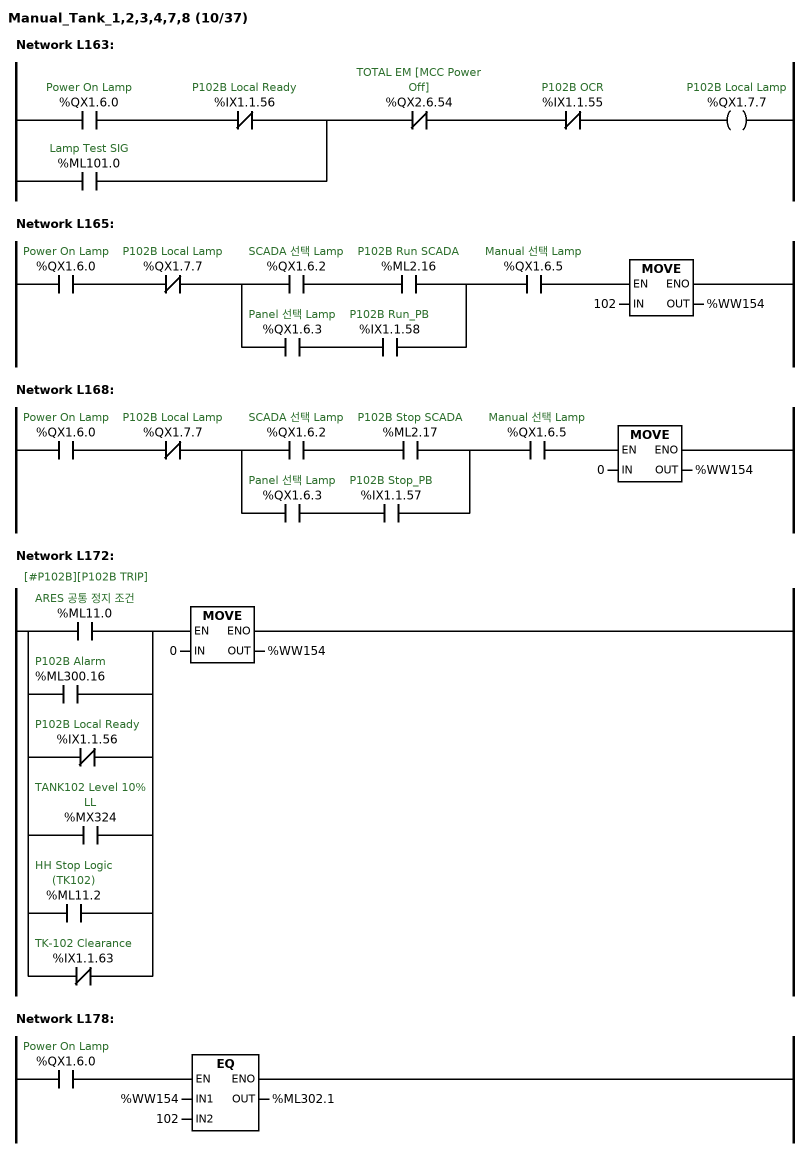
(* [picture p24: Manual_Tank_1,2,3,4,7,8 rungs L163-L178] *)
(* Rung L163 *)
%QX1.7.7 := ((%QX1.6.0 AND NOT %IX1.1.56) OR %ML101.0) AND NOT %QX2.6.54 AND NOT %IX1.1.55;
(* Rung L165 *)
IF %QX1.6.0 AND NOT %QX1.7.7 AND ((%QX1.6.2 AND %ML2.16) OR (%QX1.6.3 AND %IX1.1.58)) AND %QX1.6.5 THEN
    %WW154 := 102;
END_IF;
(* Rung L168 *)
IF %QX1.6.0 AND NOT %QX1.7.7 AND ((%QX1.6.2 AND %ML2.17) OR (%QX1.6.3 AND %IX1.1.57)) AND %QX1.6.5 THEN
    %WW154 := 0;
END_IF;
(* [#P102B][P102B TRIP] *)
(* Rung L172 *)
IF %ML11.0 OR %ML300.16 OR NOT %IX1.1.56 OR %MX324 OR %ML11.2 OR NOT %IX1.1.63 THEN %WW154 := 0; END_IF;
(* Rung L178 *)
IF %QX1.6.0 THEN %ML302.1 := %WW154 = 102; END_IF;

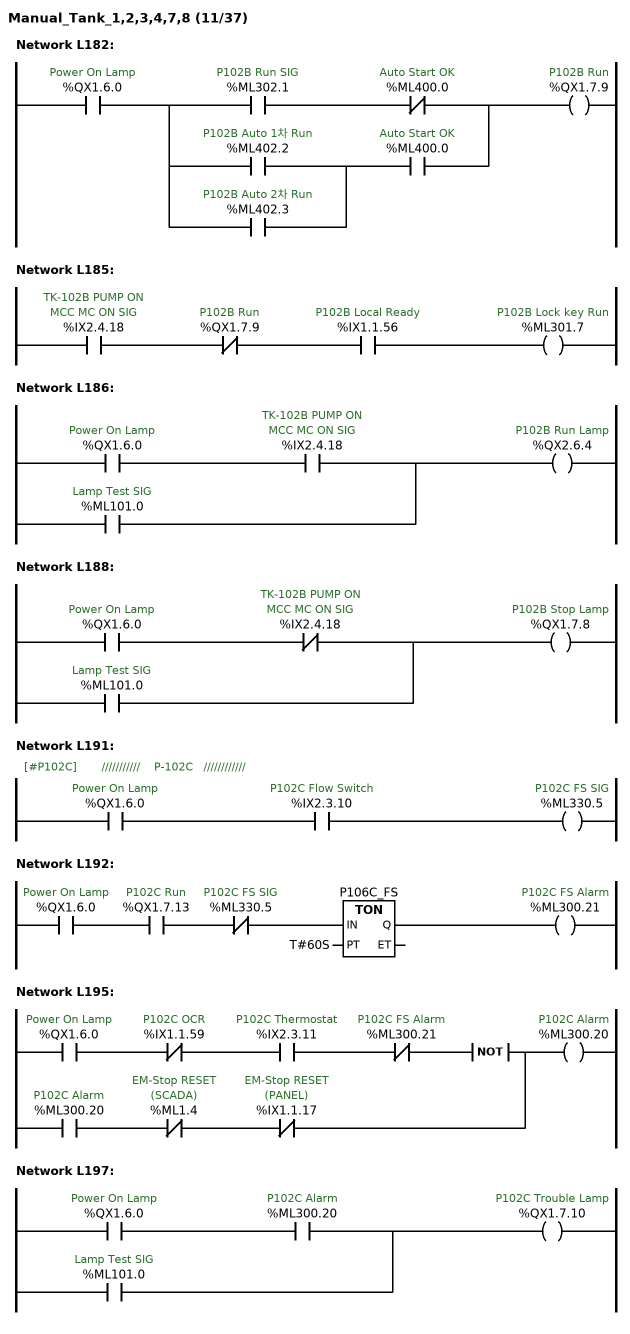
(* Rung L182 *)
%QX1.7.9 := %QX1.6.0 AND ((%ML302.1 AND NOT %ML400.0) OR ((%ML402.2 OR %ML402.3) AND %ML400.0));
(* Rung L185 *)
%ML301.7 := %IX2.4.18 AND NOT %QX1.7.9 AND %IX1.1.56;
(* Rung L186 *)
%QX2.6.4 := (%QX1.6.0 AND %IX2.4.18) OR %ML101.0;
(* Rung L188 *)
%QX1.7.8 := (%QX1.6.0 AND NOT %IX2.4.18) OR %ML101.0;
(* [#P102C]       ///////////    P-102C   //////////// *)
(* Rung L191 *)
%ML330.5 := %QX1.6.0 AND %IX2.3.10;
(* Rung L192 *)
P106C_FS(IN := %QX1.6.0 AND %QX1.7.13 AND NOT %ML330.5, PT := T#60S);
%ML300.21 := P106C_FS.Q;
(* Rung L195 *)
%ML300.20 := NOT (%QX1.6.0 AND NOT %IX1.1.59 AND %IX2.3.11 AND NOT %ML300.21) OR (%ML300.20 AND NOT %ML1.4 AND NOT %IX1.1.17);
(* Rung L197 *)
%QX1.7.10 := (%QX1.6.0 AND %ML300.20) OR %ML101.0;

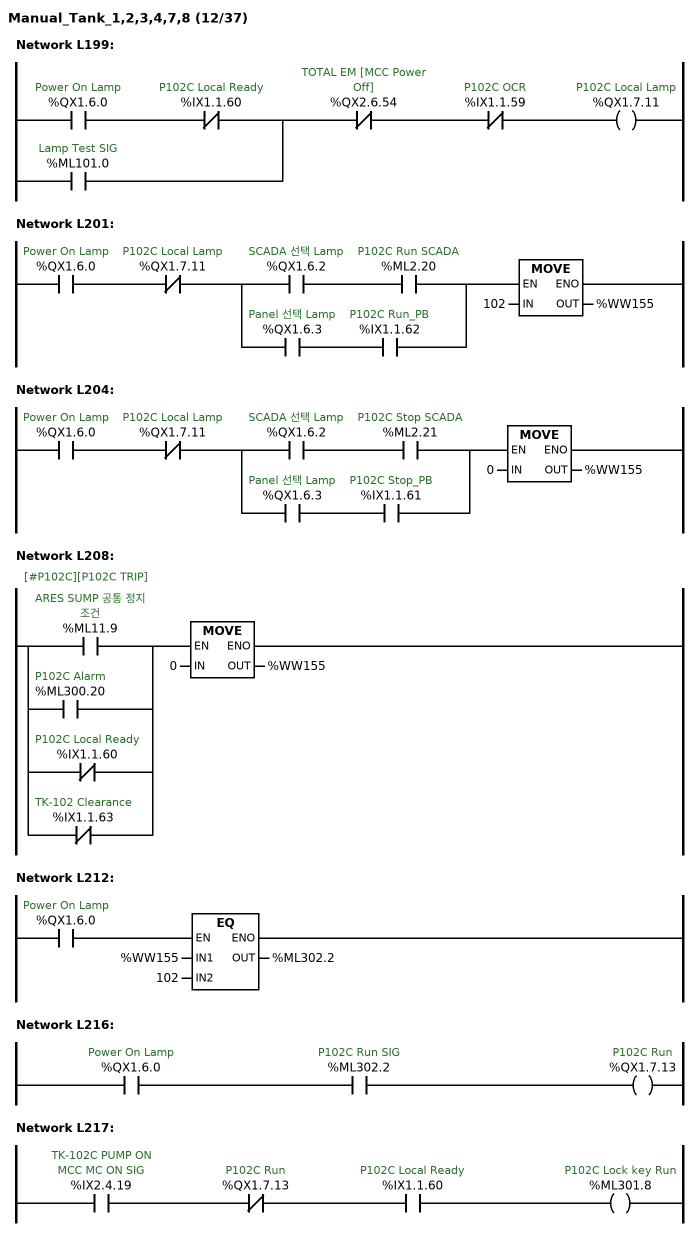
(* Rung L199 *)
%QX1.7.11 := ((%QX1.6.0 AND NOT %IX1.1.60) OR %ML101.0) AND NOT %QX2.6.54 AND NOT %IX1.1.59;
(* Rung L201 *)
IF %QX1.6.0 AND NOT %QX1.7.11 AND ((%QX1.6.2 AND %ML2.20) OR (%QX1.6.3 AND %IX1.1.62)) THEN
    %WW155 := 102;
END_IF;
(* Rung L204 *)
IF %QX1.6.0 AND NOT %QX1.7.11 AND ((%QX1.6.2 AND %ML2.21) OR (%QX1.6.3 AND %IX1.1.61)) THEN
    %WW155 := 0;
END_IF;
(* [#P102C][P102C TRIP] *)
(* Rung L208 *)
IF %ML11.9 OR %ML300.20 OR NOT %IX1.1.60 OR NOT %IX1.1.63 THEN %WW155 := 0; END_IF;
(* Rung L212 *)
IF %QX1.6.0 THEN %ML302.2 := %WW155 = 102; END_IF;
(* Rung L216 *)
%QX1.7.13 := %QX1.6.0 AND %ML302.2;
(* Rung L217 *)
%ML301.8 := %IX2.4.19 AND NOT %QX1.7.13 AND %IX1.1.60;

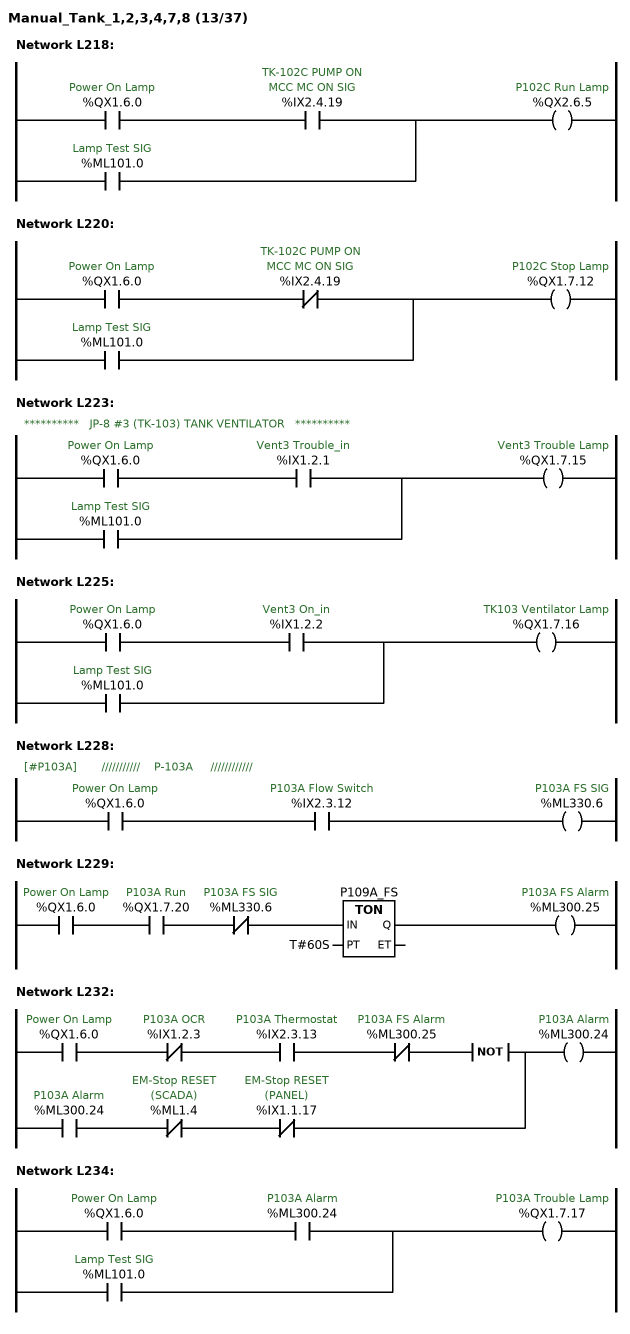
(* Rung L218 *)
%QX2.6.5 := (%QX1.6.0 AND %IX2.4.19) OR %ML101.0;
(* Rung L220 *)
%QX1.7.12 := (%QX1.6.0 AND NOT %IX2.4.19) OR %ML101.0;
(* **********   JP-8 #3 (TK-103) TANK VENTILATOR   ********** *)
(* Rung L223 *)
%QX1.7.15 := (%QX1.6.0 AND %IX1.2.1) OR %ML101.0;
(* Rung L225 *)
%QX1.7.16 := (%QX1.6.0 AND %IX1.2.2) OR %ML101.0;
(* [#P103A]       ///////////    P-103A     //////////// *)
(* Rung L228 *)
%ML330.6 := %QX1.6.0 AND %IX2.3.12;
(* Rung L229 *)
P109A_FS(IN := %QX1.6.0 AND %QX1.7.20 AND NOT %ML330.6, PT := T#60S);
%ML300.25 := P109A_FS.Q;
(* Rung L232 *)
%ML300.24 := NOT (%QX1.6.0 AND NOT %IX1.2.3 AND %IX2.3.13 AND NOT %ML300.25) OR (%ML300.24 AND NOT %ML1.4 AND NOT %IX1.1.17);
(* Rung L234 *)
%QX1.7.17 := (%QX1.6.0 AND %ML300.24) OR %ML101.0;

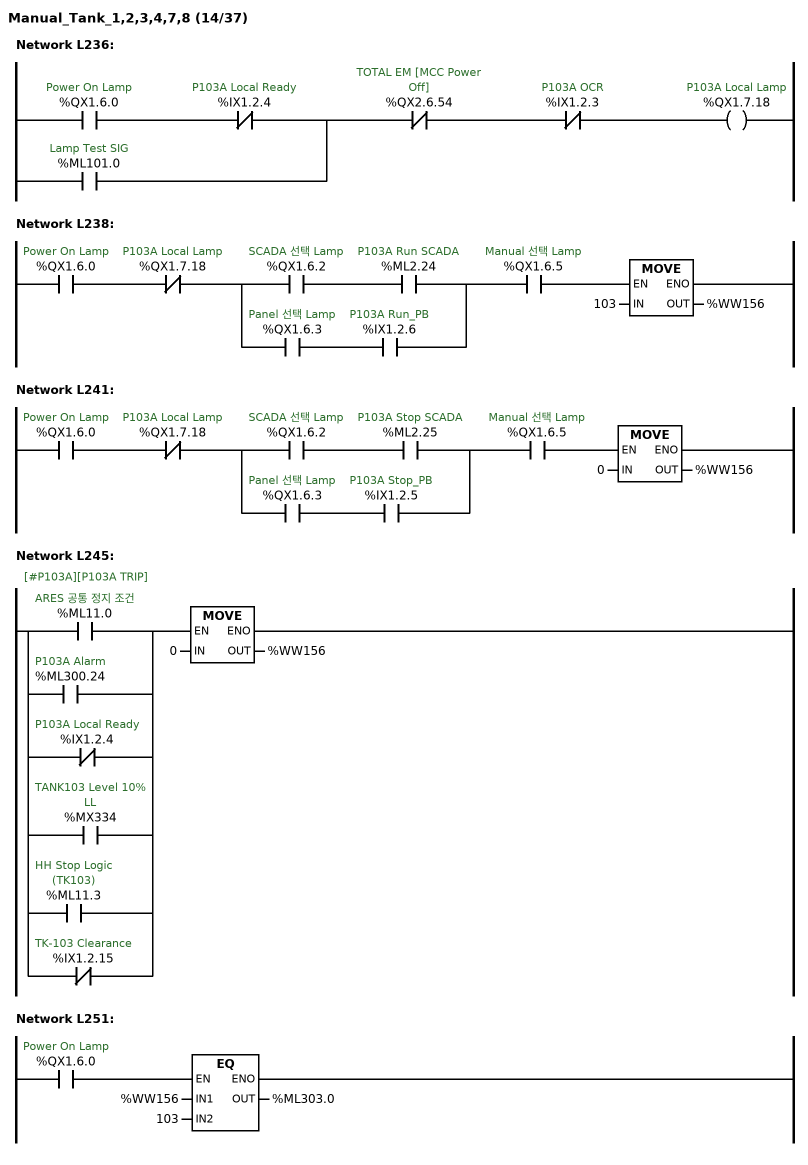
(* Rung L236 *)
%QX1.7.18 := ((%QX1.6.0 AND NOT %IX1.2.4) OR %ML101.0) AND NOT %QX2.6.54 AND NOT %IX1.2.3;
(* Rung L238 *)
IF %QX1.6.0 AND NOT %QX1.7.18 AND ((%QX1.6.2 AND %ML2.24) OR (%QX1.6.3 AND %IX1.2.6)) AND %QX1.6.5 THEN
    %WW156 := 103;
END_IF;
(* Rung L241 *)
IF %QX1.6.0 AND NOT %QX1.7.18 AND ((%QX1.6.2 AND %ML2.25) OR (%QX1.6.3 AND %IX1.2.5)) AND %QX1.6.5 THEN
    %WW156 := 0;
END_IF;
(* [#P103A][P103A TRIP] *)
(* Rung L245 *)
IF %ML11.0 OR %ML300.24 OR NOT %IX1.2.4 OR %MX334 OR %ML11.3 OR NOT %IX1.2.15 THEN %WW156 := 0; END_IF;
(* Rung L251 *)
IF %QX1.6.0 THEN %ML303.0 := %WW156 = 103; END_IF;

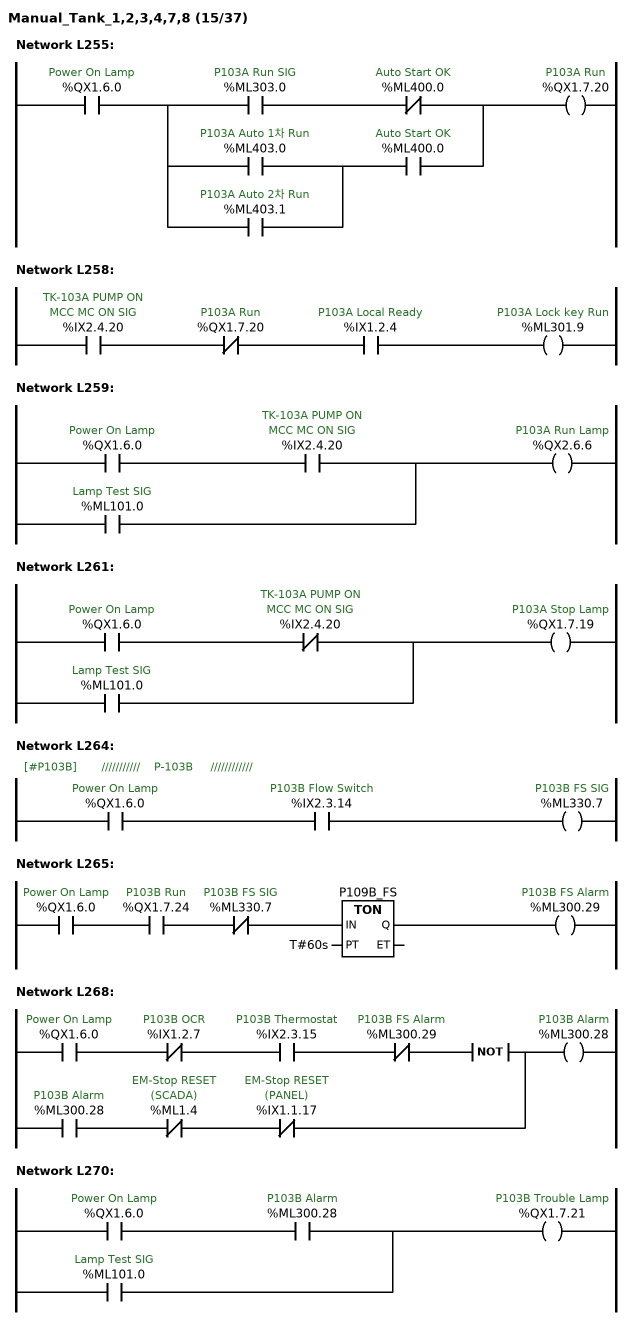
(* Rung L255 *)
%QX1.7.20 := %QX1.6.0 AND ((%ML303.0 AND NOT %ML400.0) OR ((%ML403.0 OR %ML403.1) AND %ML400.0));
(* Rung L258 *)
%ML301.9 := %IX2.4.20 AND NOT %QX1.7.20 AND %IX1.2.4;
(* Rung L259 *)
%QX2.6.6 := (%QX1.6.0 AND %IX2.4.20) OR %ML101.0;
(* Rung L261 *)
%QX1.7.19 := (%QX1.6.0 AND NOT %IX2.4.20) OR %ML101.0;
(* [#P103B]       ///////////    P-103B     //////////// *)
(* Rung L264 *)
%ML330.7 := %QX1.6.0 AND %IX2.3.14;
(* Rung L265 *)
P109B_FS(IN := %QX1.6.0 AND %QX1.7.24 AND NOT %ML330.7, PT := T#60s);
%ML300.29 := P109B_FS.Q;
(* Rung L268 *)
%ML300.28 := NOT (%QX1.6.0 AND NOT %IX1.2.7 AND %IX2.3.15 AND NOT %ML300.29) OR (%ML300.28 AND NOT %ML1.4 AND NOT %IX1.1.17);
(* Rung L270 *)
%QX1.7.21 := (%QX1.6.0 AND %ML300.28) OR %ML101.0;

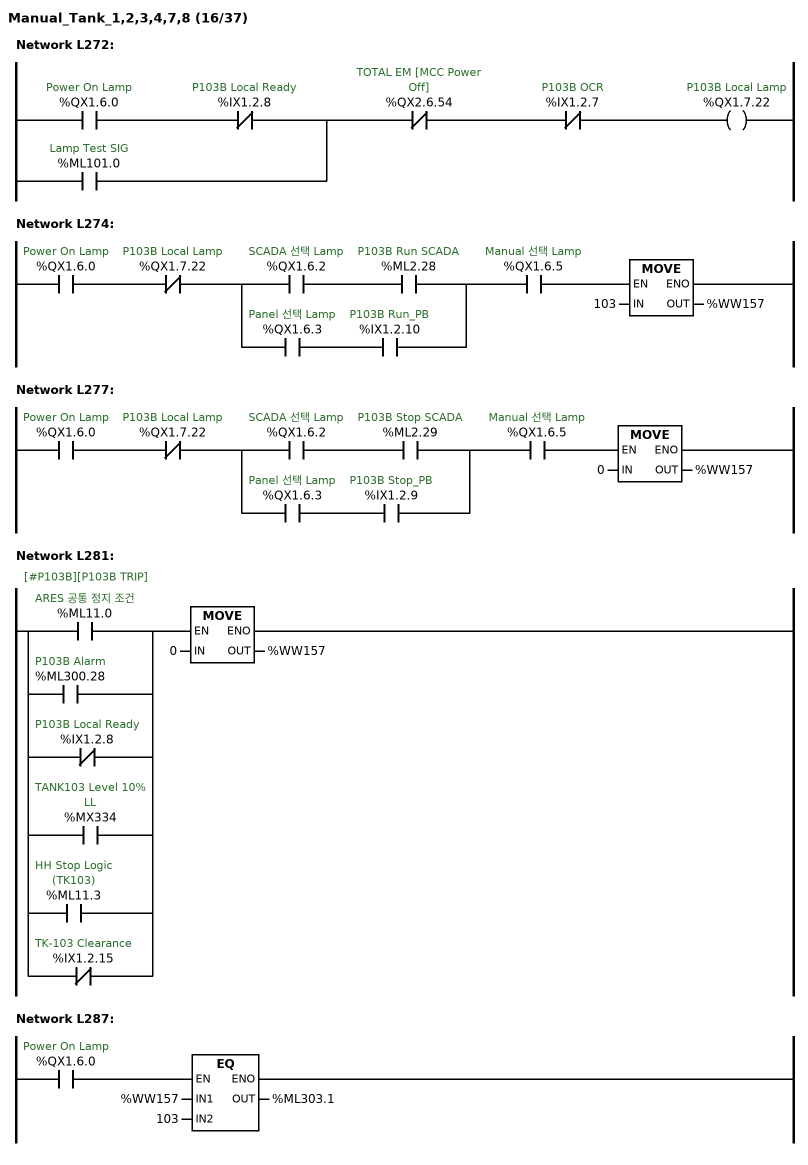
(* Rung L272 *)
%QX1.7.22 := ((%QX1.6.0 AND NOT %IX1.2.8) OR %ML101.0) AND NOT %QX2.6.54 AND NOT %IX1.2.7;
(* Rung L274 *)
IF %QX1.6.0 AND NOT %QX1.7.22 AND ((%QX1.6.2 AND %ML2.28) OR (%QX1.6.3 AND %IX1.2.10)) AND %QX1.6.5 THEN
    %WW157 := 103;
END_IF;
(* Rung L277 *)
IF %QX1.6.0 AND NOT %QX1.7.22 AND ((%QX1.6.2 AND %ML2.29) OR (%QX1.6.3 AND %IX1.2.9)) AND %QX1.6.5 THEN
    %WW157 := 0;
END_IF;
(* [#P103B][P103B TRIP] *)
(* Rung L281 *)
IF %ML11.0 OR %ML300.28 OR NOT %IX1.2.8 OR %MX334 OR %ML11.3 OR NOT %IX1.2.15 THEN %WW157 := 0; END_IF;
(* Rung L287 *)
IF %QX1.6.0 THEN %ML303.1 := %WW157 = 103; END_IF;

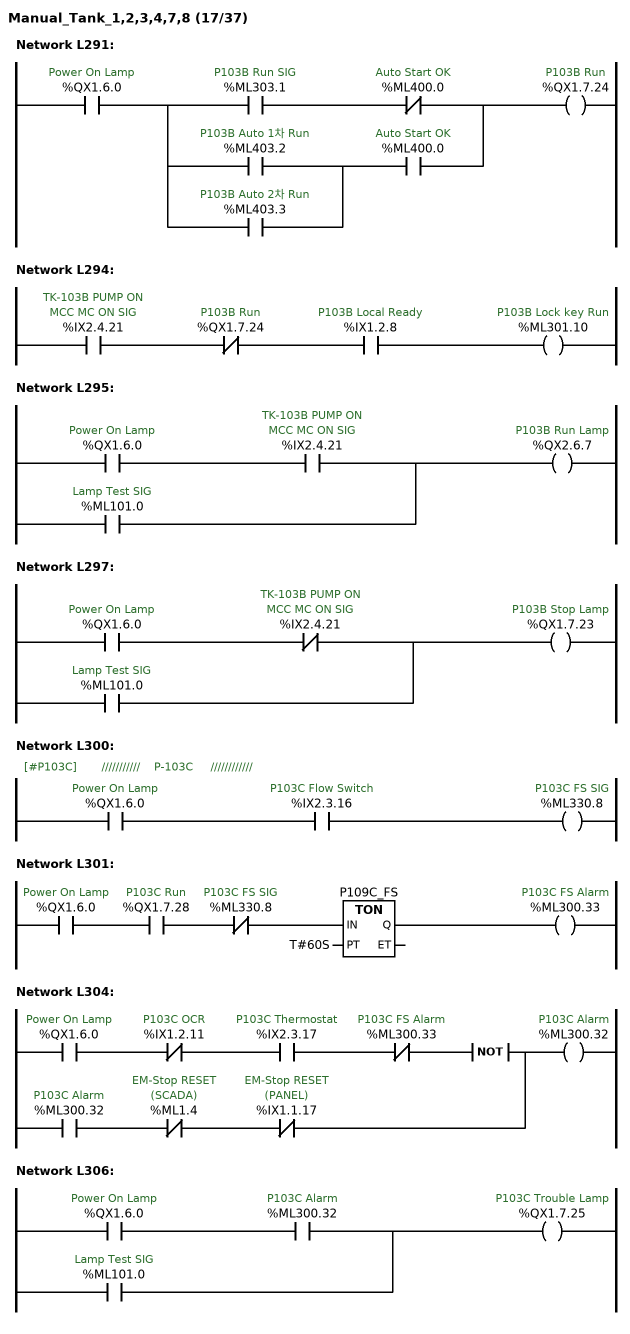
(* Rung L291 *)
%QX1.7.24 := %QX1.6.0 AND ((%ML303.1 AND NOT %ML400.0) OR ((%ML403.2 OR %ML403.3) AND %ML400.0));
(* Rung L294 *)
%ML301.10 := %IX2.4.21 AND NOT %QX1.7.24 AND %IX1.2.8;
(* Rung L295 *)
%QX2.6.7 := (%QX1.6.0 AND %IX2.4.21) OR %ML101.0;
(* Rung L297 *)
%QX1.7.23 := (%QX1.6.0 AND NOT %IX2.4.21) OR %ML101.0;
(* [#P103C]       ///////////    P-103C     //////////// *)
(* Rung L300 *)
%ML330.8 := %QX1.6.0 AND %IX2.3.16;
(* Rung L301 *)
P109C_FS(IN := %QX1.6.0 AND %QX1.7.28 AND NOT %ML330.8, PT := T#60S);
%ML300.33 := P109C_FS.Q;
(* Rung L304 *)
%ML300.32 := NOT (%QX1.6.0 AND NOT %IX1.2.11 AND %IX2.3.17 AND NOT %ML300.33) OR (%ML300.32 AND NOT %ML1.4 AND NOT %IX1.1.17);
(* Rung L306 *)
%QX1.7.25 := (%QX1.6.0 AND %ML300.32) OR %ML101.0;

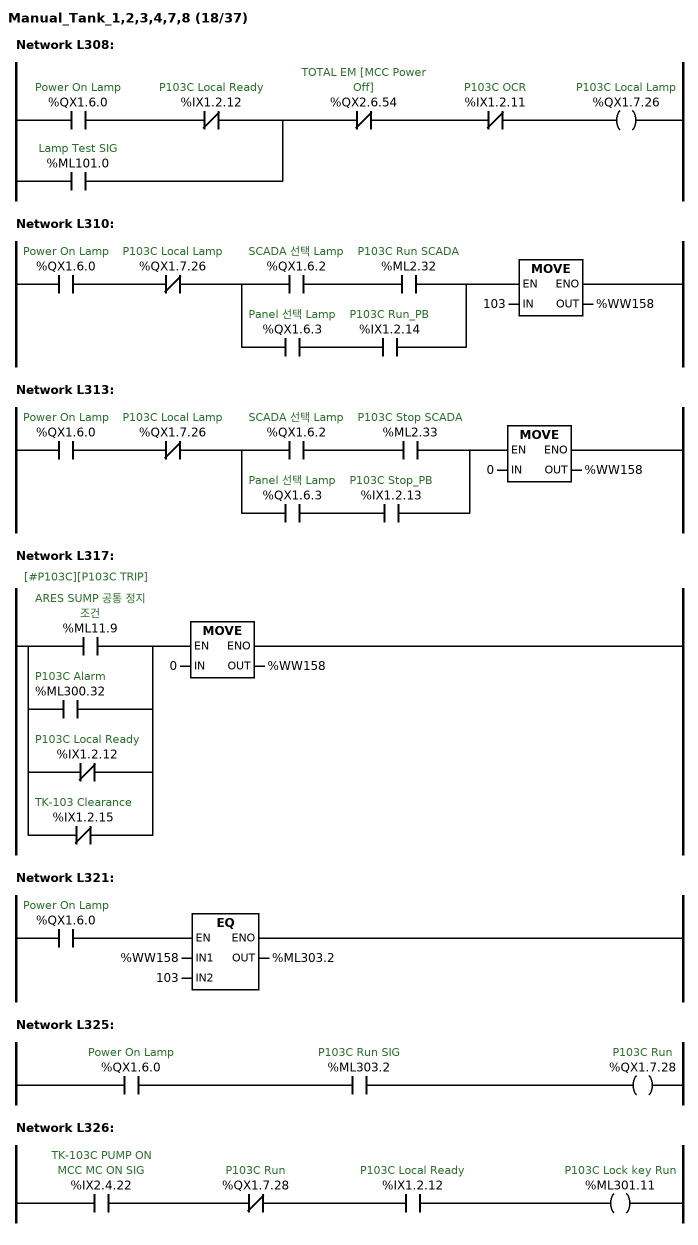
(* Rung L308 *)
%QX1.7.26 := ((%QX1.6.0 AND NOT %IX1.2.12) OR %ML101.0) AND NOT %QX2.6.54 AND NOT %IX1.2.11;
(* Rung L310 *)
IF %QX1.6.0 AND NOT %QX1.7.26 AND ((%QX1.6.2 AND %ML2.32) OR (%QX1.6.3 AND %IX1.2.14)) THEN
    %WW158 := 103;
END_IF;
(* Rung L313 *)
IF %QX1.6.0 AND NOT %QX1.7.26 AND ((%QX1.6.2 AND %ML2.33) OR (%QX1.6.3 AND %IX1.2.13)) THEN
    %WW158 := 0;
END_IF;
(* [#P103C][P103C TRIP] *)
(* Rung L317 *)
IF %ML11.9 OR %ML300.32 OR NOT %IX1.2.12 OR NOT %IX1.2.15 THEN %WW158 := 0; END_IF;
(* Rung L321 *)
IF %QX1.6.0 THEN %ML303.2 := %WW158 = 103; END_IF;
(* Rung L325 *)
%QX1.7.28 := %QX1.6.0 AND %ML303.2;
(* Rung L326 *)
%ML301.11 := %IX2.4.22 AND NOT %QX1.7.28 AND %IX1.2.12;

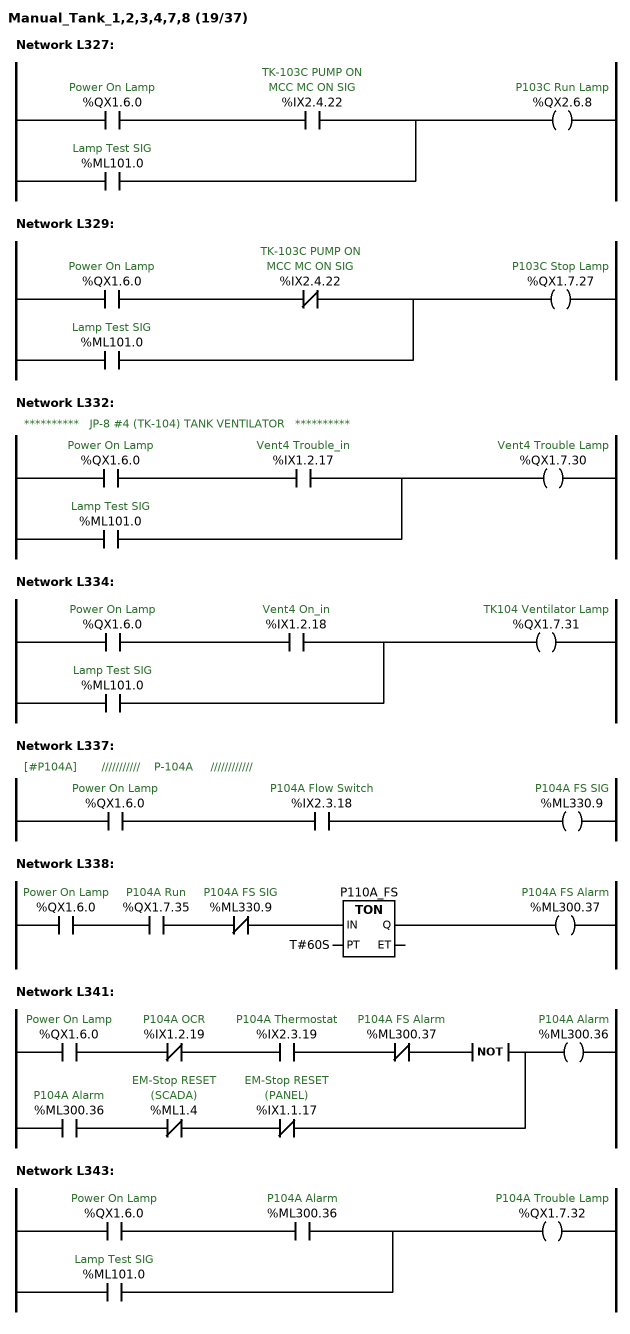
(* Rung L327 *)
%QX2.6.8 := (%QX1.6.0 AND %IX2.4.22) OR %ML101.0;
(* Rung L329 *)
%QX1.7.27 := (%QX1.6.0 AND NOT %IX2.4.22) OR %ML101.0;
(* **********   JP-8 #4 (TK-104) TANK VENTILATOR   ********** *)
(* Rung L332 *)
%QX1.7.30 := (%QX1.6.0 AND %IX1.2.17) OR %ML101.0;
(* Rung L334 *)
%QX1.7.31 := (%QX1.6.0 AND %IX1.2.18) OR %ML101.0;
(* [#P104A]       ///////////    P-104A     //////////// *)
(* Rung L337 *)
%ML330.9 := %QX1.6.0 AND %IX2.3.18;
(* Rung L338 *)
P110A_FS(IN := %QX1.6.0 AND %QX1.7.35 AND NOT %ML330.9, PT := T#60S);
%ML300.37 := P110A_FS.Q;
(* Rung L341 *)
%ML300.36 := NOT (%QX1.6.0 AND NOT %IX1.2.19 AND %IX2.3.19 AND NOT %ML300.37) OR (%ML300.36 AND NOT %ML1.4 AND NOT %IX1.1.17);
(* Rung L343 *)
%QX1.7.32 := (%QX1.6.0 AND %ML300.36) OR %ML101.0;

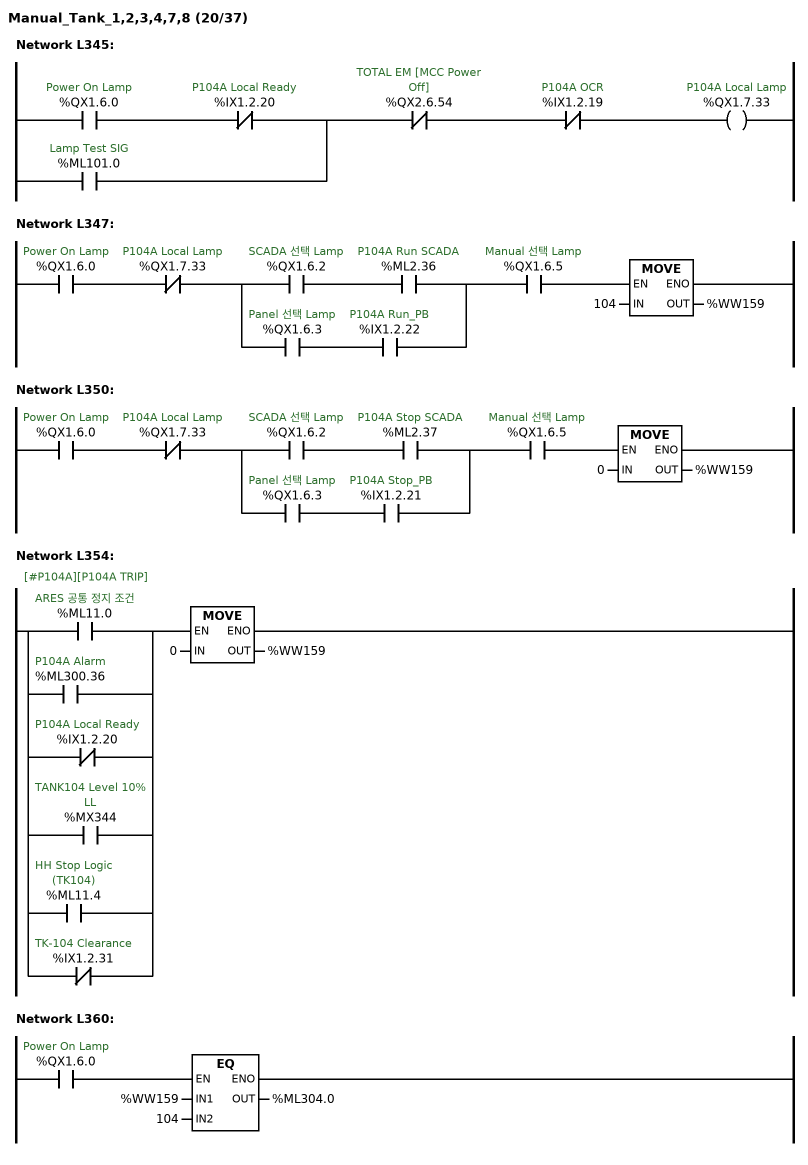
(* Rung L345 *)
%QX1.7.33 := ((%QX1.6.0 AND NOT %IX1.2.20) OR %ML101.0) AND NOT %QX2.6.54 AND NOT %IX1.2.19;
(* Rung L347 *)
IF %QX1.6.0 AND NOT %QX1.7.33 AND ((%QX1.6.2 AND %ML2.36) OR (%QX1.6.3 AND %IX1.2.22)) AND %QX1.6.5 THEN
    %WW159 := 104;
END_IF;
(* Rung L350 *)
IF %QX1.6.0 AND NOT %QX1.7.33 AND ((%QX1.6.2 AND %ML2.37) OR (%QX1.6.3 AND %IX1.2.21)) AND %QX1.6.5 THEN
    %WW159 := 0;
END_IF;
(* [#P104A][P104A TRIP] *)
(* Rung L354 *)
IF %ML11.0 OR %ML300.36 OR NOT %IX1.2.20 OR %MX344 OR %ML11.4 OR NOT %IX1.2.31 THEN %WW159 := 0; END_IF;
(* Rung L360 *)
IF %QX1.6.0 THEN %ML304.0 := %WW159 = 104; END_IF;

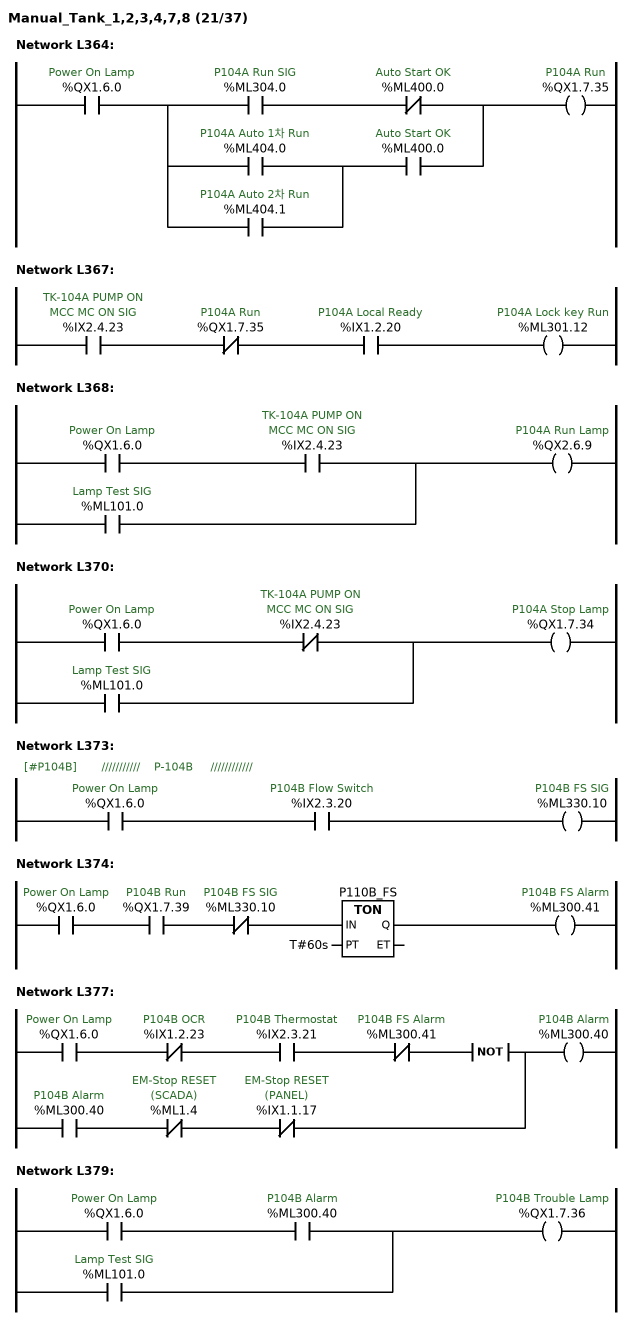
(* Rung L364 *)
%QX1.7.35 := %QX1.6.0 AND ((%ML304.0 AND NOT %ML400.0) OR ((%ML404.0 OR %ML404.1) AND %ML400.0));
(* Rung L367 *)
%ML301.12 := %IX2.4.23 AND NOT %QX1.7.35 AND %IX1.2.20;
(* Rung L368 *)
%QX2.6.9 := (%QX1.6.0 AND %IX2.4.23) OR %ML101.0;
(* Rung L370 *)
%QX1.7.34 := (%QX1.6.0 AND NOT %IX2.4.23) OR %ML101.0;
(* [#P104B]       ///////////    P-104B     //////////// *)
(* Rung L373 *)
%ML330.10 := %QX1.6.0 AND %IX2.3.20;
(* Rung L374 *)
P110B_FS(IN := %QX1.6.0 AND %QX1.7.39 AND NOT %ML330.10, PT := T#60s);
%ML300.41 := P110B_FS.Q;
(* Rung L377 *)
%ML300.40 := NOT (%QX1.6.0 AND NOT %IX1.2.23 AND %IX2.3.21 AND NOT %ML300.41) OR (%ML300.40 AND NOT %ML1.4 AND NOT %IX1.1.17);
(* Rung L379 *)
%QX1.7.36 := (%QX1.6.0 AND %ML300.40) OR %ML101.0;

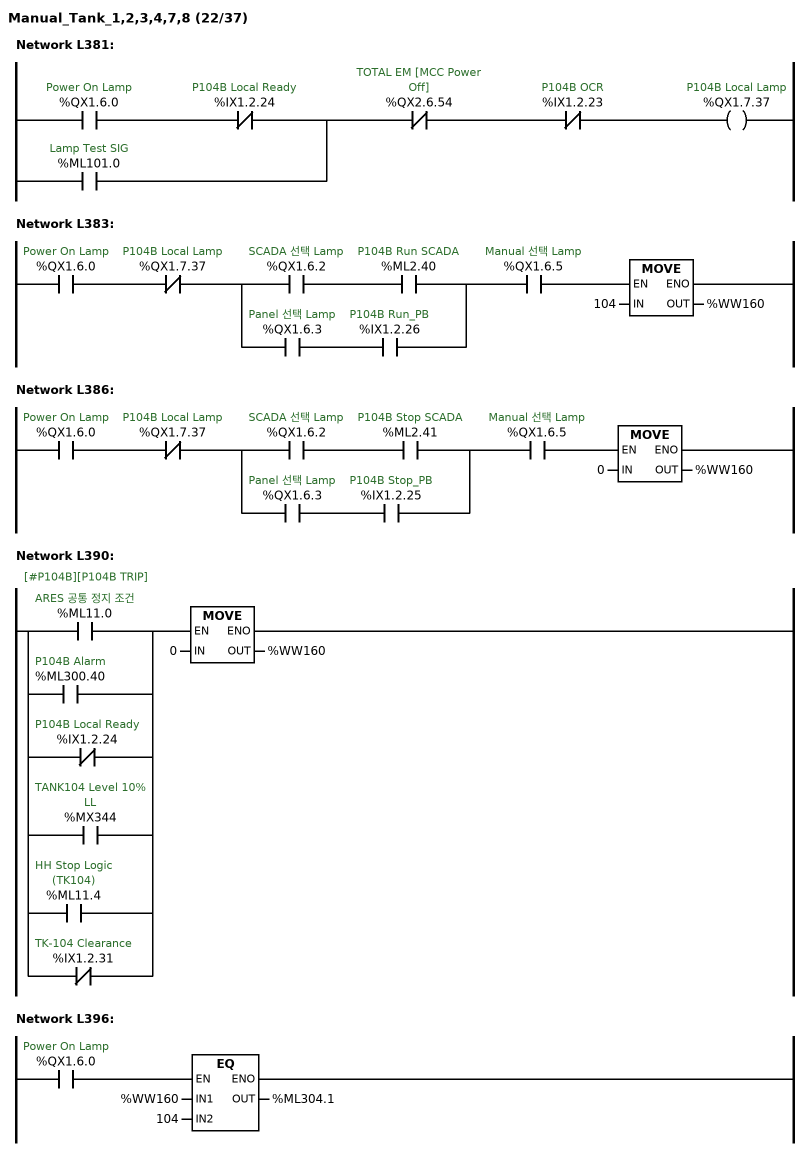
(* Rung L381 *)
%QX1.7.37 := ((%QX1.6.0 AND NOT %IX1.2.24) OR %ML101.0) AND NOT %QX2.6.54 AND NOT %IX1.2.23;
(* Rung L383 *)
IF %QX1.6.0 AND NOT %QX1.7.37 AND ((%QX1.6.2 AND %ML2.40) OR (%QX1.6.3 AND %IX1.2.26)) AND %QX1.6.5 THEN
    %WW160 := 104;
END_IF;
(* Rung L386 *)
IF %QX1.6.0 AND NOT %QX1.7.37 AND ((%QX1.6.2 AND %ML2.41) OR (%QX1.6.3 AND %IX1.2.25)) AND %QX1.6.5 THEN
    %WW160 := 0;
END_IF;
(* [#P104B][P104B TRIP] *)
(* Rung L390 *)
IF %ML11.0 OR %ML300.40 OR NOT %IX1.2.24 OR %MX344 OR %ML11.4 OR NOT %IX1.2.31 THEN %WW160 := 0; END_IF;
(* Rung L396 *)
IF %QX1.6.0 THEN %ML304.1 := %WW160 = 104; END_IF;

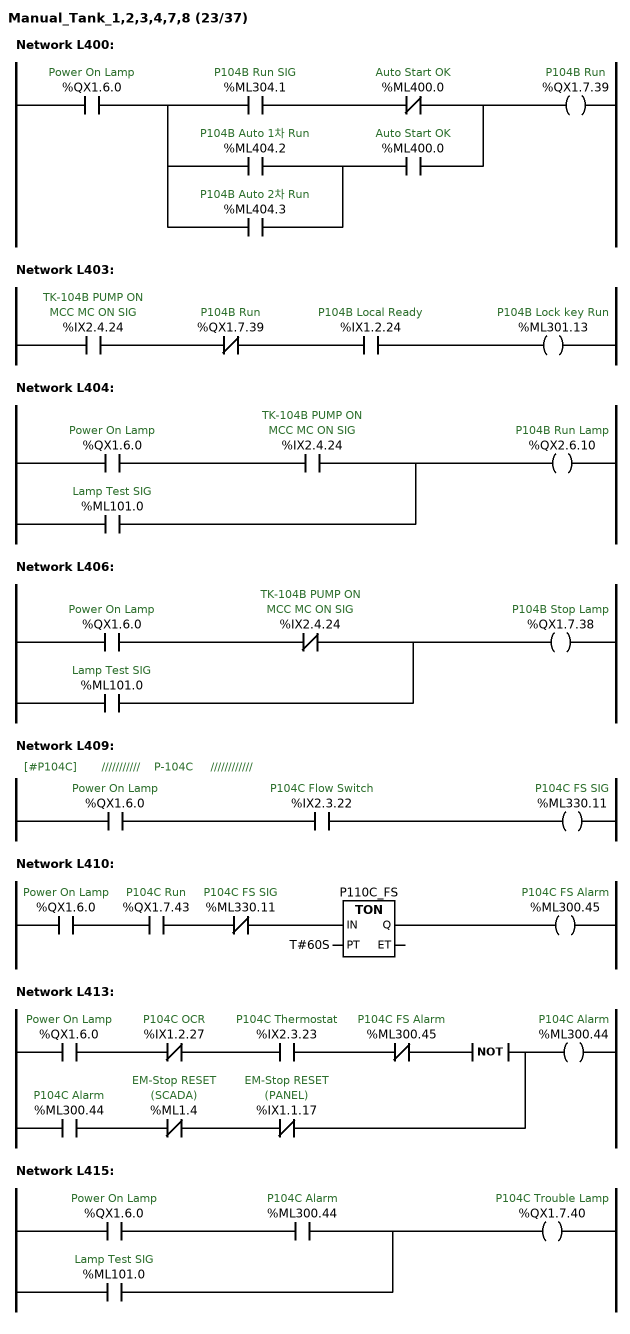
(* Rung L400 *)
%QX1.7.39 := %QX1.6.0 AND ((%ML304.1 AND NOT %ML400.0) OR ((%ML404.2 OR %ML404.3) AND %ML400.0));
(* Rung L403 *)
%ML301.13 := %IX2.4.24 AND NOT %QX1.7.39 AND %IX1.2.24;
(* Rung L404 *)
%QX2.6.10 := (%QX1.6.0 AND %IX2.4.24) OR %ML101.0;
(* Rung L406 *)
%QX1.7.38 := (%QX1.6.0 AND NOT %IX2.4.24) OR %ML101.0;
(* [#P104C]       ///////////    P-104C     //////////// *)
(* Rung L409 *)
%ML330.11 := %QX1.6.0 AND %IX2.3.22;
(* Rung L410 *)
P110C_FS(IN := %QX1.6.0 AND %QX1.7.43 AND NOT %ML330.11, PT := T#60S);
%ML300.45 := P110C_FS.Q;
(* Rung L413 *)
%ML300.44 := NOT (%QX1.6.0 AND NOT %IX1.2.27 AND %IX2.3.23 AND NOT %ML300.45) OR (%ML300.44 AND NOT %ML1.4 AND NOT %IX1.1.17);
(* Rung L415 *)
%QX1.7.40 := (%QX1.6.0 AND %ML300.44) OR %ML101.0;

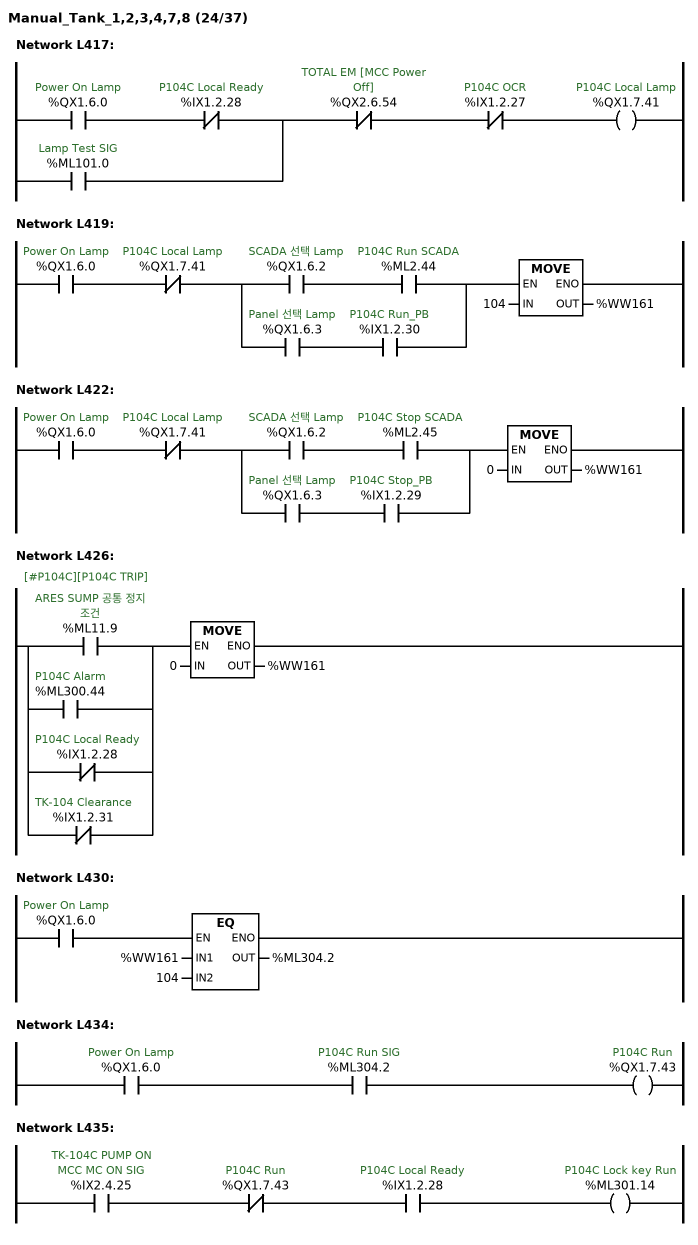
(* Rung L417 *)
%QX1.7.41 := ((%QX1.6.0 AND NOT %IX1.2.28) OR %ML101.0) AND NOT %QX2.6.54 AND NOT %IX1.2.27;
(* Rung L419 *)
IF %QX1.6.0 AND NOT %QX1.7.41 AND ((%QX1.6.2 AND %ML2.44) OR (%QX1.6.3 AND %IX1.2.30)) THEN
    %WW161 := 104;
END_IF;
(* Rung L422 *)
IF %QX1.6.0 AND NOT %QX1.7.41 AND ((%QX1.6.2 AND %ML2.45) OR (%QX1.6.3 AND %IX1.2.29)) THEN
    %WW161 := 0;
END_IF;
(* [#P104C][P104C TRIP] *)
(* Rung L426 *)
IF %ML11.9 OR %ML300.44 OR NOT %IX1.2.28 OR NOT %IX1.2.31 THEN %WW161 := 0; END_IF;
(* Rung L430 *)
IF %QX1.6.0 THEN %ML304.2 := %WW161 = 104; END_IF;
(* Rung L434 *)
%QX1.7.43 := %QX1.6.0 AND %ML304.2;
(* Rung L435 *)
%ML301.14 := %IX2.4.25 AND NOT %QX1.7.43 AND %IX1.2.28;

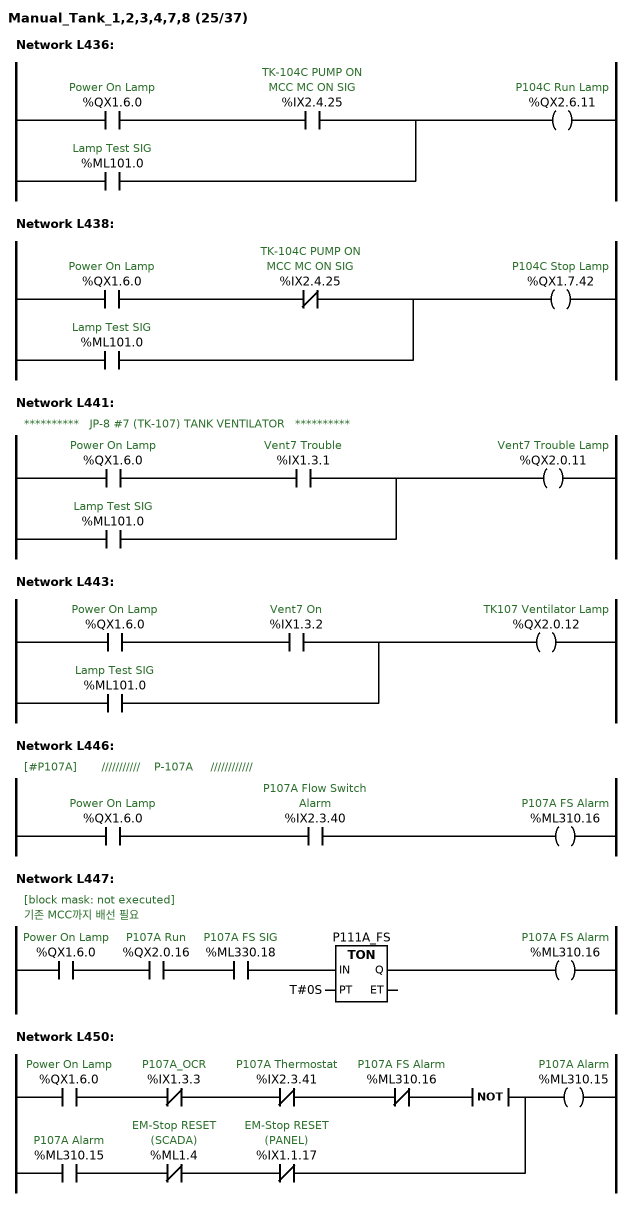
(* Rung L436 *)
%QX2.6.11 := (%QX1.6.0 AND %IX2.4.25) OR %ML101.0;
(* Rung L438 *)
%QX1.7.42 := (%QX1.6.0 AND NOT %IX2.4.25) OR %ML101.0;
(* **********   JP-8 #7 (TK-107) TANK VENTILATOR   ********** *)
(* Rung L441 *)
%QX2.0.11 := (%QX1.6.0 AND %IX1.3.1) OR %ML101.0;
(* Rung L443 *)
%QX2.0.12 := (%QX1.6.0 AND %IX1.3.2) OR %ML101.0;
(* [#P107A]       ///////////    P-107A     //////////// *)
(* Rung L446 *)
%ML310.16 := %QX1.6.0 AND %IX2.3.40;
(* Rung L447 is block-masked: not executed *)
// P111A_FS(IN := %QX1.6.0 AND %QX2.0.16 AND %ML330.18, PT := T#0S);
// %ML310.16 := P111A_FS.Q;
(* 기존 MCC까지 배선 필요 *)
(* Rung L450 *)
%ML310.15 := NOT (%QX1.6.0 AND NOT %IX1.3.3 AND NOT %IX2.3.41 AND NOT %ML310.16) OR (%ML310.15 AND NOT %ML1.4 AND NOT %IX1.1.17);

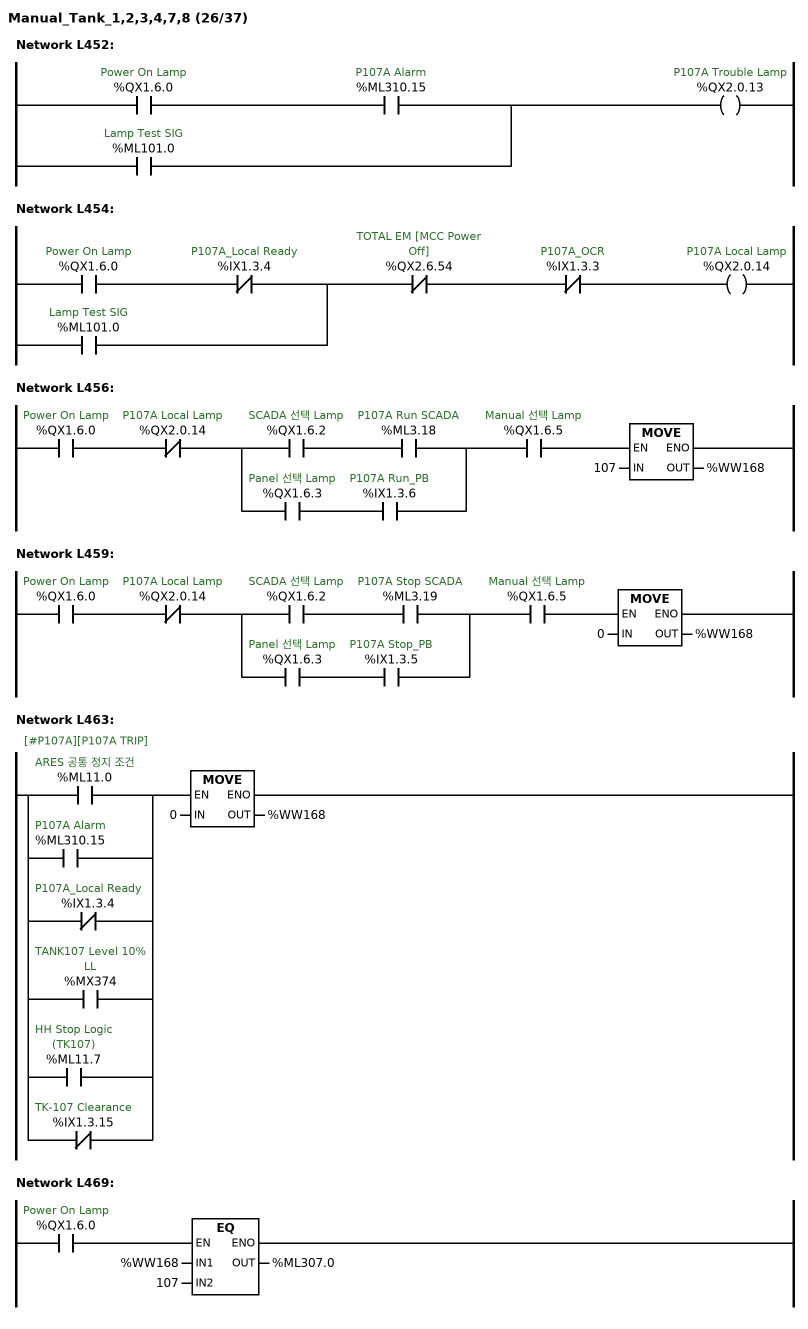
(* Rung L452 *)
%QX2.0.13 := (%QX1.6.0 AND %ML310.15) OR %ML101.0;
(* Rung L454 *)
%QX2.0.14 := ((%QX1.6.0 AND NOT %IX1.3.4) OR %ML101.0) AND NOT %QX2.6.54 AND NOT %IX1.3.3;
(* Rung L456 *)
IF %QX1.6.0 AND NOT %QX2.0.14 AND ((%QX1.6.2 AND %ML3.18) OR (%QX1.6.3 AND %IX1.3.6)) AND %QX1.6.5 THEN
    %WW168 := 107;
END_IF;
(* Rung L459 *)
IF %QX1.6.0 AND NOT %QX2.0.14 AND ((%QX1.6.2 AND %ML3.19) OR (%QX1.6.3 AND %IX1.3.5)) AND %QX1.6.5 THEN
    %WW168 := 0;
END_IF;
(* [#P107A][P107A TRIP] *)
(* Rung L463 *)
IF %ML11.0 OR %ML310.15 OR NOT %IX1.3.4 OR %MX374 OR %ML11.7 OR NOT %IX1.3.15 THEN %WW168 := 0; END_IF;
(* Rung L469 *)
IF %QX1.6.0 THEN %ML307.0 := %WW168 = 107; END_IF;

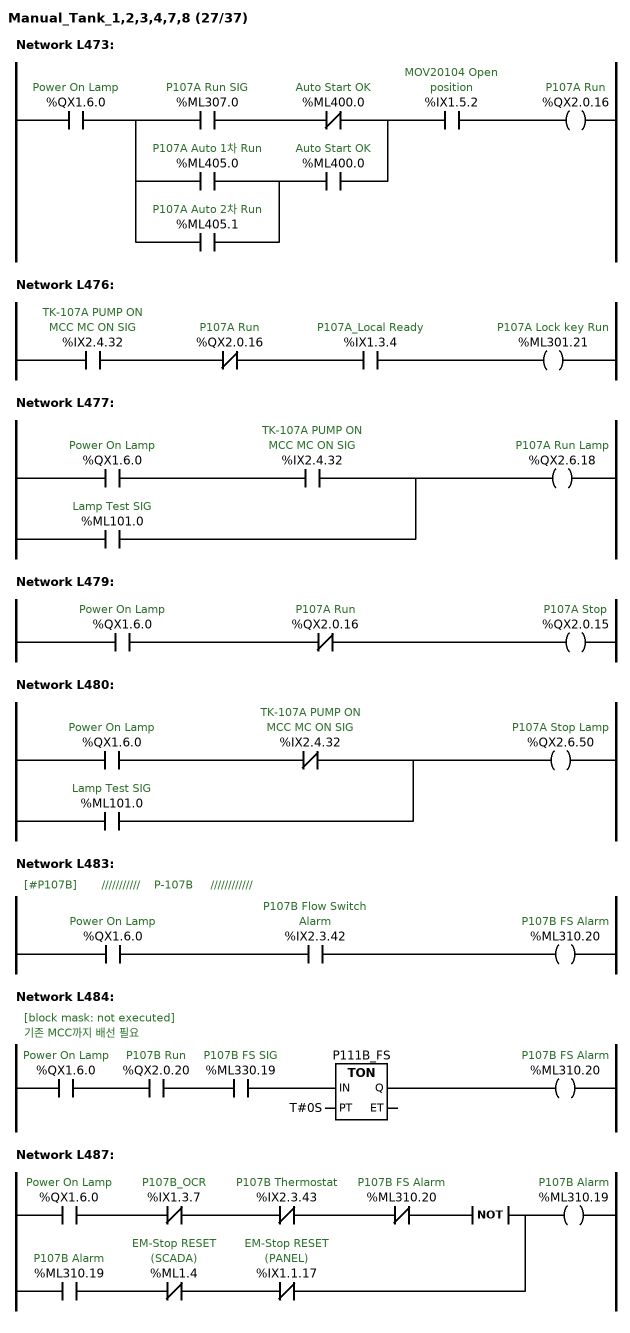
(* Rung L473 *)
%QX2.0.16 := %QX1.6.0 AND ((%ML307.0 AND NOT %ML400.0) OR ((%ML405.0 OR %ML405.1) AND %ML400.0)) AND %IX1.5.2;
(* Rung L476 *)
%ML301.21 := %IX2.4.32 AND NOT %QX2.0.16 AND %IX1.3.4;
(* Rung L477 *)
%QX2.6.18 := (%QX1.6.0 AND %IX2.4.32) OR %ML101.0;
(* Rung L479 *)
%QX2.0.15 := %QX1.6.0 AND NOT %QX2.0.16;
(* Rung L480 *)
%QX2.6.50 := (%QX1.6.0 AND NOT %IX2.4.32) OR %ML101.0;
(* [#P107B]       ///////////    P-107B     //////////// *)
(* Rung L483 *)
%ML310.20 := %QX1.6.0 AND %IX2.3.42;
(* Rung L484 is block-masked: not executed *)
// P111B_FS(IN := %QX1.6.0 AND %QX2.0.20 AND %ML330.19, PT := T#0S);
// %ML310.20 := P111B_FS.Q;
(* 기존 MCC까지 배선 필요 *)
(* Rung L487 *)
%ML310.19 := NOT (%QX1.6.0 AND NOT %IX1.3.7 AND NOT %IX2.3.43 AND NOT %ML310.20) OR (%ML310.19 AND NOT %ML1.4 AND NOT %IX1.1.17);

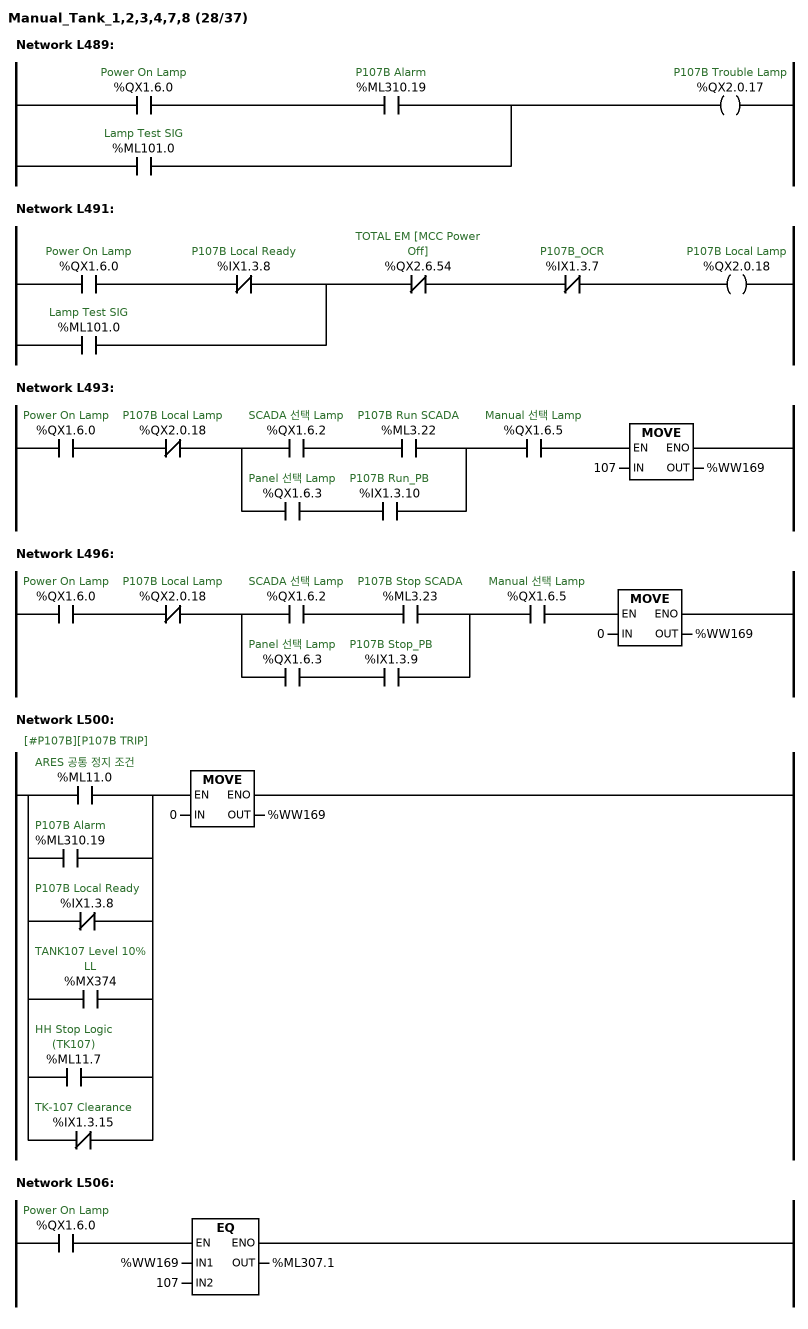
(* Rung L489 *)
%QX2.0.17 := (%QX1.6.0 AND %ML310.19) OR %ML101.0;
(* Rung L491 *)
%QX2.0.18 := ((%QX1.6.0 AND NOT %IX1.3.8) OR %ML101.0) AND NOT %QX2.6.54 AND NOT %IX1.3.7;
(* Rung L493 *)
IF %QX1.6.0 AND NOT %QX2.0.18 AND ((%QX1.6.2 AND %ML3.22) OR (%QX1.6.3 AND %IX1.3.10)) AND %QX1.6.5 THEN
    %WW169 := 107;
END_IF;
(* Rung L496 *)
IF %QX1.6.0 AND NOT %QX2.0.18 AND ((%QX1.6.2 AND %ML3.23) OR (%QX1.6.3 AND %IX1.3.9)) AND %QX1.6.5 THEN
    %WW169 := 0;
END_IF;
(* [#P107B][P107B TRIP] *)
(* Rung L500 *)
IF %ML11.0 OR %ML310.19 OR NOT %IX1.3.8 OR %MX374 OR %ML11.7 OR NOT %IX1.3.15 THEN %WW169 := 0; END_IF;
(* Rung L506 *)
IF %QX1.6.0 THEN %ML307.1 := %WW169 = 107; END_IF;

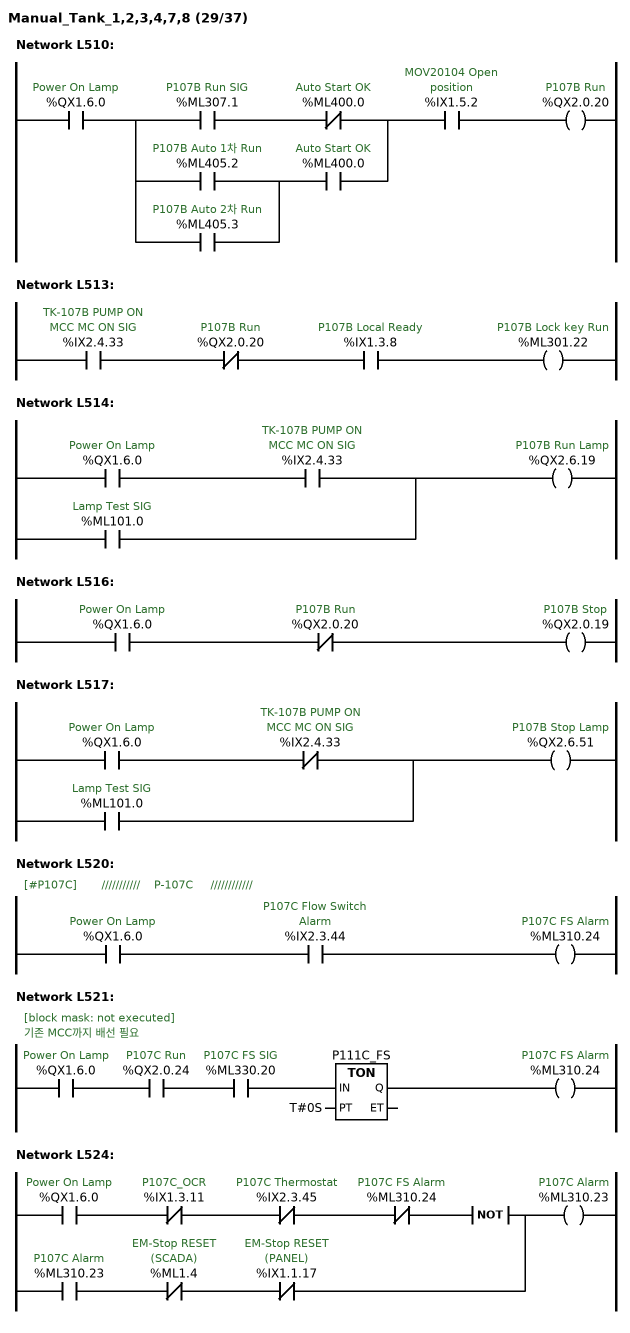
(* Rung L510 *)
%QX2.0.20 := %QX1.6.0 AND ((%ML307.1 AND NOT %ML400.0) OR ((%ML405.2 OR %ML405.3) AND %ML400.0)) AND %IX1.5.2;
(* Rung L513 *)
%ML301.22 := %IX2.4.33 AND NOT %QX2.0.20 AND %IX1.3.8;
(* Rung L514 *)
%QX2.6.19 := (%QX1.6.0 AND %IX2.4.33) OR %ML101.0;
(* Rung L516 *)
%QX2.0.19 := %QX1.6.0 AND NOT %QX2.0.20;
(* Rung L517 *)
%QX2.6.51 := (%QX1.6.0 AND NOT %IX2.4.33) OR %ML101.0;
(* [#P107C]       ///////////    P-107C     //////////// *)
(* Rung L520 *)
%ML310.24 := %QX1.6.0 AND %IX2.3.44;
(* Rung L521 is block-masked: not executed *)
// P111C_FS(IN := %QX1.6.0 AND %QX2.0.24 AND %ML330.20, PT := T#0S);
// %ML310.24 := P111C_FS.Q;
(* 기존 MCC까지 배선 필요 *)
(* Rung L524 *)
%ML310.23 := NOT (%QX1.6.0 AND NOT %IX1.3.11 AND NOT %IX2.3.45 AND NOT %ML310.24) OR (%ML310.23 AND NOT %ML1.4 AND NOT %IX1.1.17);

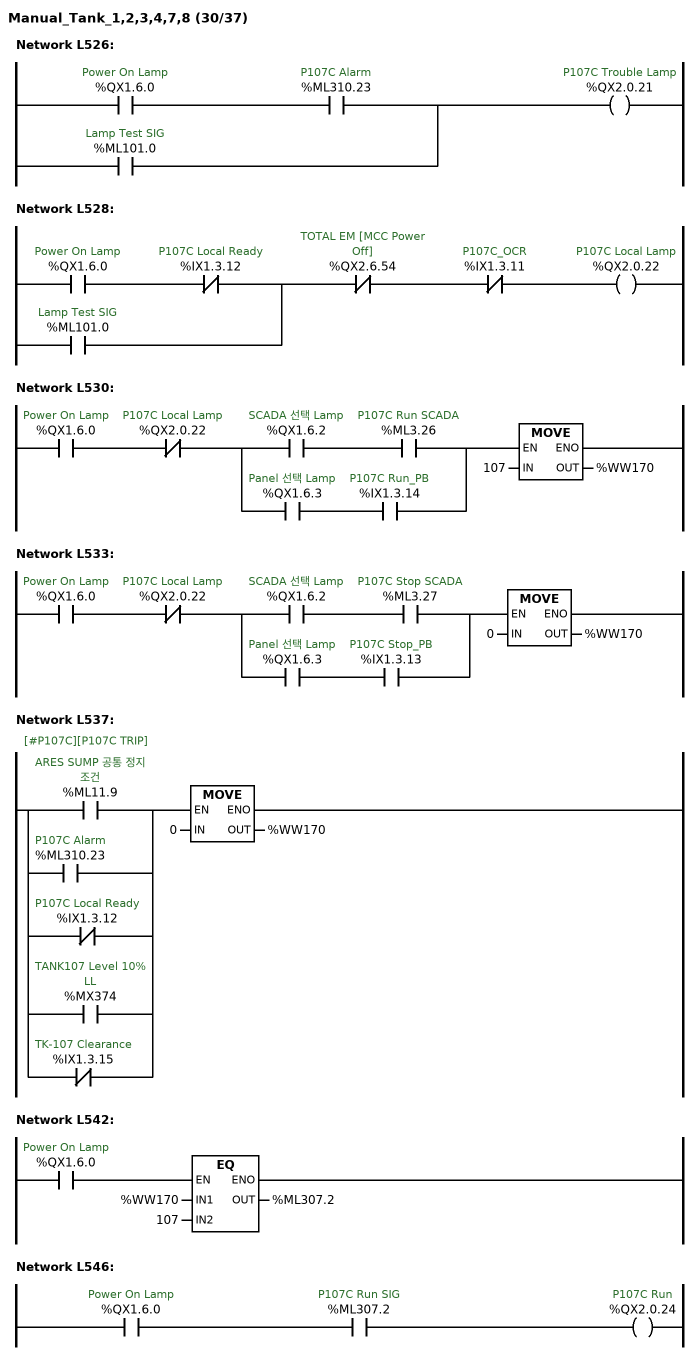
(* Rung L526 *)
%QX2.0.21 := (%QX1.6.0 AND %ML310.23) OR %ML101.0;
(* Rung L528 *)
%QX2.0.22 := ((%QX1.6.0 AND NOT %IX1.3.12) OR %ML101.0) AND NOT %QX2.6.54 AND NOT %IX1.3.11;
(* Rung L530 *)
IF %QX1.6.0 AND NOT %QX2.0.22 AND ((%QX1.6.2 AND %ML3.26) OR (%QX1.6.3 AND %IX1.3.14)) THEN
    %WW170 := 107;
END_IF;
(* Rung L533 *)
IF %QX1.6.0 AND NOT %QX2.0.22 AND ((%QX1.6.2 AND %ML3.27) OR (%QX1.6.3 AND %IX1.3.13)) THEN
    %WW170 := 0;
END_IF;
(* [#P107C][P107C TRIP] *)
(* Rung L537 *)
IF %ML11.9 OR %ML310.23 OR NOT %IX1.3.12 OR %MX374 OR NOT %IX1.3.15 THEN %WW170 := 0; END_IF;
(* Rung L542 *)
IF %QX1.6.0 THEN %ML307.2 := %WW170 = 107; END_IF;
(* Rung L546 *)
%QX2.0.24 := %QX1.6.0 AND %ML307.2;

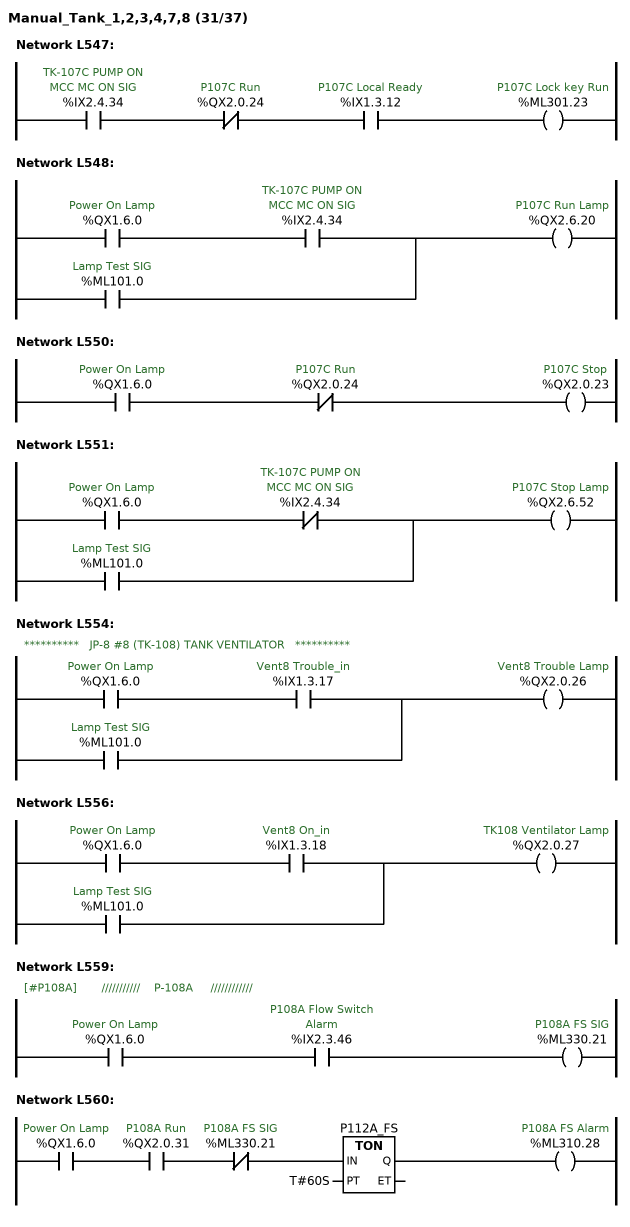
(* Rung L547 *)
%ML301.23 := %IX2.4.34 AND NOT %QX2.0.24 AND %IX1.3.12;
(* Rung L548 *)
%QX2.6.20 := (%QX1.6.0 AND %IX2.4.34) OR %ML101.0;
(* Rung L550 *)
%QX2.0.23 := %QX1.6.0 AND NOT %QX2.0.24;
(* Rung L551 *)
%QX2.6.52 := (%QX1.6.0 AND NOT %IX2.4.34) OR %ML101.0;
(* **********   JP-8 #8 (TK-108) TANK VENTILATOR   ********** *)
(* Rung L554 *)
%QX2.0.26 := (%QX1.6.0 AND %IX1.3.17) OR %ML101.0;
(* Rung L556 *)
%QX2.0.27 := (%QX1.6.0 AND %IX1.3.18) OR %ML101.0;
(* [#P108A]       ///////////    P-108A     //////////// *)
(* Rung L559 *)
%ML330.21 := %QX1.6.0 AND %IX2.3.46;
(* Rung L560 *)
P112A_FS(IN := %QX1.6.0 AND %QX2.0.31 AND NOT %ML330.21, PT := T#60S);
%ML310.28 := P112A_FS.Q;

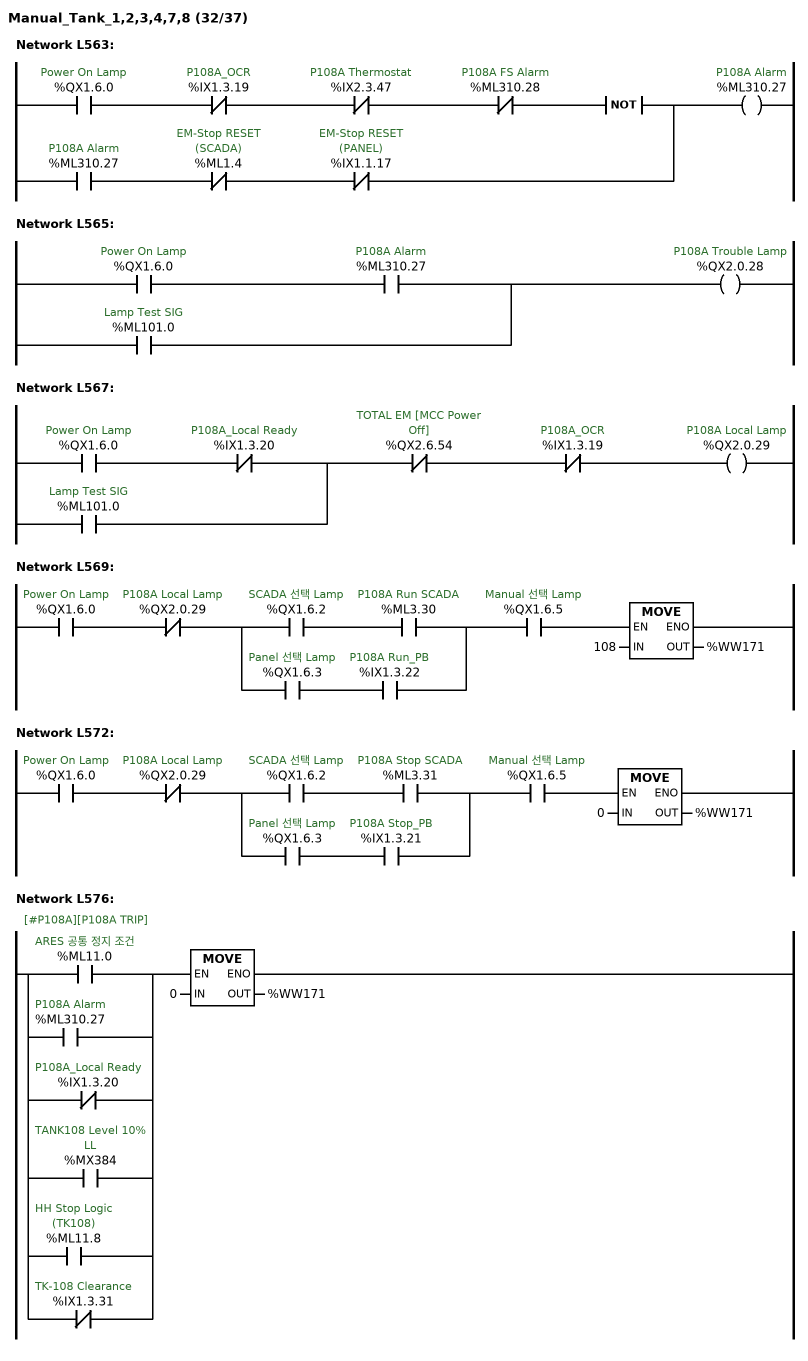
(* Rung L563 *)
%ML310.27 := NOT (%QX1.6.0 AND NOT %IX1.3.19 AND NOT %IX2.3.47 AND NOT %ML310.28) OR (%ML310.27 AND NOT %ML1.4 AND NOT %IX1.1.17);
(* Rung L565 *)
%QX2.0.28 := (%QX1.6.0 AND %ML310.27) OR %ML101.0;
(* Rung L567 *)
%QX2.0.29 := ((%QX1.6.0 AND NOT %IX1.3.20) OR %ML101.0) AND NOT %QX2.6.54 AND NOT %IX1.3.19;
(* Rung L569 *)
IF %QX1.6.0 AND NOT %QX2.0.29 AND ((%QX1.6.2 AND %ML3.30) OR (%QX1.6.3 AND %IX1.3.22)) AND %QX1.6.5 THEN
    %WW171 := 108;
END_IF;
(* Rung L572 *)
IF %QX1.6.0 AND NOT %QX2.0.29 AND ((%QX1.6.2 AND %ML3.31) OR (%QX1.6.3 AND %IX1.3.21)) AND %QX1.6.5 THEN
    %WW171 := 0;
END_IF;
(* [#P108A][P108A TRIP] *)
(* Rung L576 *)
IF %ML11.0 OR %ML310.27 OR NOT %IX1.3.20 OR %MX384 OR %ML11.8 OR NOT %IX1.3.31 THEN %WW171 := 0; END_IF;

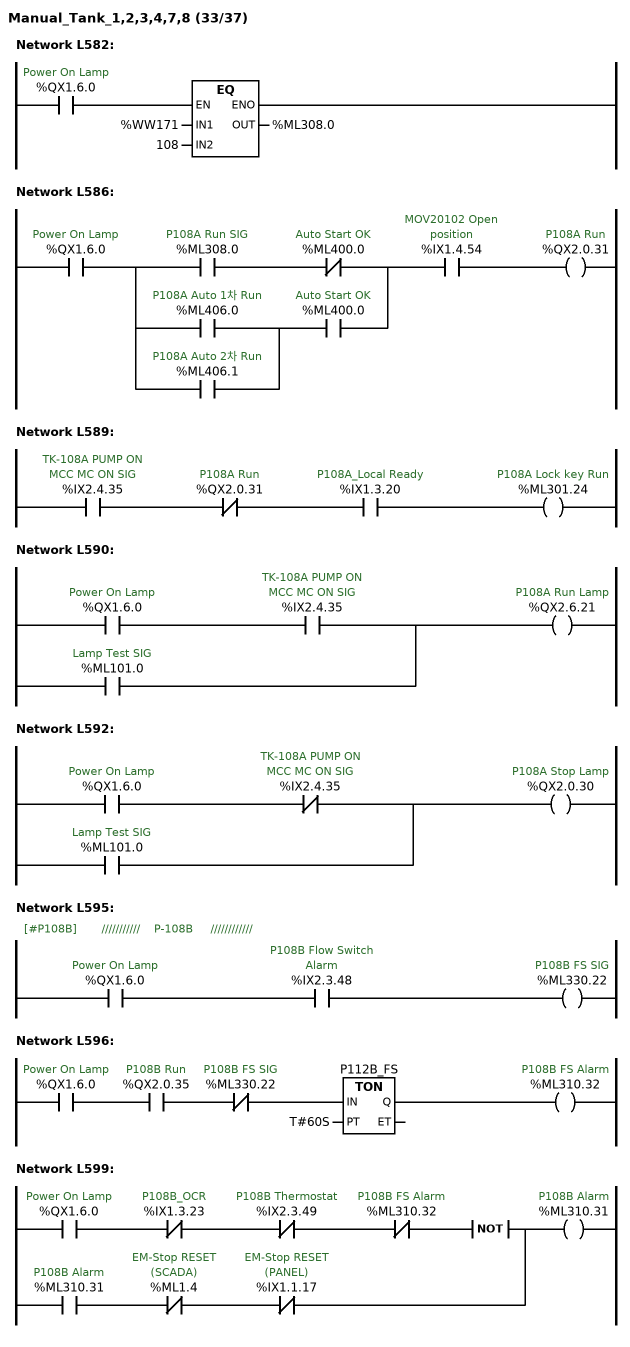
(* Rung L582 *)
IF %QX1.6.0 THEN %ML308.0 := %WW171 = 108; END_IF;
(* Rung L586 *)
%QX2.0.31 := %QX1.6.0 AND ((%ML308.0 AND NOT %ML400.0) OR ((%ML406.0 OR %ML406.1) AND %ML400.0)) AND %IX1.4.54;
(* Rung L589 *)
%ML301.24 := %IX2.4.35 AND NOT %QX2.0.31 AND %IX1.3.20;
(* Rung L590 *)
%QX2.6.21 := (%QX1.6.0 AND %IX2.4.35) OR %ML101.0;
(* Rung L592 *)
%QX2.0.30 := (%QX1.6.0 AND NOT %IX2.4.35) OR %ML101.0;
(* [#P108B]       ///////////    P-108B     //////////// *)
(* Rung L595 *)
%ML330.22 := %QX1.6.0 AND %IX2.3.48;
(* Rung L596 *)
P112B_FS(IN := %QX1.6.0 AND %QX2.0.35 AND NOT %ML330.22, PT := T#60S);
%ML310.32 := P112B_FS.Q;
(* Rung L599 *)
%ML310.31 := NOT (%QX1.6.0 AND NOT %IX1.3.23 AND NOT %IX2.3.49 AND NOT %ML310.32) OR (%ML310.31 AND NOT %ML1.4 AND NOT %IX1.1.17);

